// TIA Portal V18 export
TYPE "SubProcessParameterP030_ShW"
// stored: IsFailsafeCompliant false
   STRUCT
      Screwing : Array[1..12] of Struct
         Torque : Real;
         Angle : Int;
         "Counter" : Int;
         Result : Int;
         NG_code : String[9];
      END_STRUCT;
   END_STRUCT;
END_TYPE
